(*udt (user defined type) of Emhart TE 1500 Profibus Based Stud:
	auth. Jessy Underhill; 
	Jan 2020; version 1.0*)


TYPE udt_Emhart_TE1500_Input :
	STRUCT
		(*Status Of Profibus Slave*)
		Inputs:udt_ProfiNode_Status;
		(*Input Bytes*)
		Byte0: BYTE;
		Byte1: BYTE;
		Byte2: BYTE;
		Byte3: BYTE;
		Byte4: BYTE;
		Byte5: BYTE;
		Byte6: BYTE;
		Byte7: BYTE;
	END_STRUCT
END_TYPE

(* stored: Version 1.1.0.1, ProductVersion 3.1.4024.5
   DUT udt_Emhart_TE1500_Input: Id {1c934b07-f495-440e-9f36-2a49959948d4} *)
